// Machine parameters - persistent, writable from PRG_Params, read everywhere.
// Defaults match the "Machine Parameters" screen in the spec.
//   *** marks values the spec left open ("??"/"X"); tune on the machine. ***
{attribute 'qualified_only'}
VAR_GLOBAL PERSISTENT
    // ===== sequence timers (HMI "Machine Parameters" page) =====
    tDewaterTime       : TIME := T#4S;     // T1 - dewater / suck slurry            [operator]
    tSPXMaxOpenTime    : TIME := T#500MS;  // T2 - SPX valve must report OPEN  within this  [engineer]
    tSPXMaxCloseTime   : TIME := T#500MS;  // T6 - SPX valve must report CLOSE within this  [engineer]  (HMI groups T2&T6)
    tSprayOpenTime     : TIME := T#3S;     // T3 - piston OPEN  stroke watchdog (P-close->P-open) [engineer]
    tSprayCloseTime    : TIME := T#3S;     // T4 - piston CLOSE stroke watchdog (P-open->P-close) [engineer]  (HMI groups T3&T4)
    tSPXDewaterTime    : TIME := T#10S;    // T5 - dewater after closing            [operator]

    // ===== pressure / pump (HMI "Machine Parameters" page) =====
    rSPXPressureTarget : REAL := 1.7;      // SPX target pressure [bar]
    rPumpSpeedBase     : REAL := 15.0;     // gear-pump base speed [Hz] (P-control starts here)

    // ===== thresholds & gains (engineer; not on the operator page) =====
    rSPXPressTol       : REAL := 0.1;      // |avg-target| >= this  -> "bad SPX pressure" warning
    rPumpDeadband      : REAL := 0.02;     // P-control deadband [bar]
    rPumpKp            : REAL := 2.0;      // *** P-control gain [Hz per bar] - spec: "double the difference??" ***
    rPumpHzMin         : REAL := 5.0;      // *** pump speed clamp, low  [Hz] ***
    rPumpHzMax         : REAL := 50.0;     // *** pump speed clamp, high [Hz] ***
    rLevelHigh         : REAL := 95.0;     // SPX tank: warn above [%]
    rLevelLow          : REAL := 20.0;     // SPX tank: warn below [%]
    rLevelEmpty        : REAL := 5.0;      // SPX tank: below -> stop pump & block mother release [%]
    rCircPressTol      : REAL := 0.5;      // spray-avg vs circulation-avg > this -> "adjust" message

    // ===== logging =====
    // Directory for the event log file (PRG_FileLogger).
    //   ''  -> TwinCAT boot folder of the TARGET (portable default:
    //          Windows C:\TwinCAT\3.1\Boot\ , BSD/Linux /usr/local/etc/TwinCAT/3.1/Boot/)
    //   'C:\kayma\machine1'          -> Windows dev PC
    //   '/home/Administrator/logs'   -> Linux/BSD PLC (folder must exist & be writable
    //                                   by the TwinCAT runtime user!)
    // PERSISTENT: set once per machine, survives reboots. Takes effect on the
    // next logged event - no restart needed.
    sLogDir            : STRING(255) := '';

    // TRUE  -> every sequence state transition is logged as INFO
    //          (~4 extra lines per spray cycle; great for commissioning)
    // FALSE -> only cycle start/complete, faults, resets, warnings
    bLogStateChanges   : BOOL := TRUE;
	bStatsEnable   : BOOL := TRUE;   // master switch
    tStatsRun      : TIME := T#1S;   // sample period while cycle active
    tStatsIdle     : TIME := T#2M;   // keep-alive period idle/fault
    nStatsHourFrom : INT  := 0;      // daily window; From=To=0 -> 24h
    nStatsHourTo   : INT  := 0;      // e.g. 6 & 22 -> log 06:00-21:59
END_VAR

VAR_GLOBAL CONSTANT
    // ===== factory defaults (RESET button on the params page) =====
    // One authoritative home for the default machine parameters.
    // If you retune the machine, change the defaults HERE (they should
    // normally mirror the init values of the persistent block above).
    cDefDewaterTime    : TIME := T#4S;      // T1
    cDefValveMaxTime   : TIME := T#500MS;   // T2 & T6
    cDefSprayTime      : TIME := T#3S;      // T3 & T4
    cDefSPXDewaterTime : TIME := T#10S;     // T5
    cDefPressTarget    : REAL := 1.7;       // [bar]
    cDefPumpSpeed      : REAL := 15.0;      // [Hz]
END_VAR

(* stored: Version 1.1.0.1, ProductVersion 3.1.4026.18
   GVL GVL_Param: Id {8b4f0c21-7d3e-4a96-b1c5-2e9d4f7a6310} *)
